SYSTEM System
  DEVICE DEV0 : NXT_RMTDEV
    RESOURCE RES0 : EMB_RES_ENH(PRIO := 0)
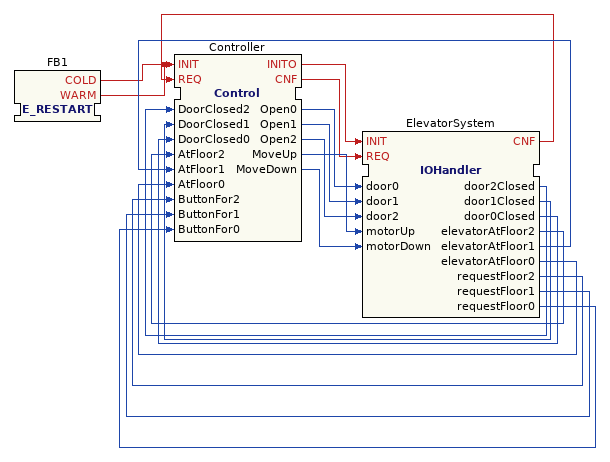
      FBS
        ElevatorSystem : IOHandler;
        FB1 : E_RESTART;
        Controller : Control;
      END_FBS
      EVENT_CONNECTIONS
        Controller.INITO TO ElevatorSystem.INIT;
        Controller.CNF TO ElevatorSystem.REQ;
        FB1.COLD TO Controller.INIT;
        FB1.WARM TO Controller.INIT;
        ElevatorSystem.CNF TO Controller.REQ;
      END_CONNECTIONS
      DATA_CONNECTIONS
        Controller.Open0 TO ElevatorSystem.door0;
        Controller.Open1 TO ElevatorSystem.door1;
        Controller.Open2 TO ElevatorSystem.door2;
        ElevatorSystem.door2Closed TO Controller.DoorClosed2;
        ElevatorSystem.door1Closed TO Controller.DoorClosed1;
        ElevatorSystem.door0Closed TO Controller.DoorClosed0;
        ElevatorSystem.elevatorAtFloor2 TO Controller.AtFloor2;
        ElevatorSystem.elevatorAtFloor1 TO Controller.AtFloor1;
        ElevatorSystem.elevatorAtFloor0 TO Controller.AtFloor0;
        ElevatorSystem.requestFloor2 TO Controller.ButtonFor2;
        ElevatorSystem.requestFloor1 TO Controller.ButtonFor1;
        ElevatorSystem.requestFloor0 TO Controller.ButtonFor0;
        Controller.MoveUp TO ElevatorSystem.motorUp;
        Controller.MoveDown TO ElevatorSystem.motorDown;
      END_CONNECTIONS
    END_RESOURCE
  END_DEVICE
END_SYSTEM
